(* Schneider Machine Expert - Basic project scelta_strategia_meccanismo, file version 3.0.0.0 *)
(* ProjectInformations: Name=Nuovo progetto *)

HARDWARE
  Cpu 0: TM221CE40R
  EthernetConfiguration: NetworkName=M221, IpAllocationMode=FixedAddress, IpAddress=0.0.0.0, SubnetMask=0.0.0.0
  SerialLineConfiguration: Baud=Baud19200, Parity=ParityEven, DataBits=DataBits8, StopBits=StopBits1, PhysicalMedium=PhysicalMediumRs485, TransmissionMode=TransmissionModeModbusRtu, SlaveId=1, Addressing=SlaveAddressing
  MastTask: UsePeriodScanMode=false, PeriodScan=100
  FastTask: Period=255
  CpuBehavior: StartingMode=StartAsPreviousState, AutoSaveRamOnEeprom=true, WatchdogPeriod=250

SYMBOLS  (address, symbol, comment, settings)
  %M5         "placeholder"
  %MW0      CONTA_PIU_UNDICI
  %MW1      CONTA_PIU_DODICI
  %MW2      CONTA_PIU_TREDICI
  %C0       CONTATORE  [Preset=100]
  %IW0.0    STRATEGIA  "11 = più undici; 12 = più dodici; 13 = più tredici;"  [Type=Type_0_10V, Scope=Scope_Normal, Minimum=0, Maximum=1000]

POU Nuovo POU
  (* SectionNumber=1 *)

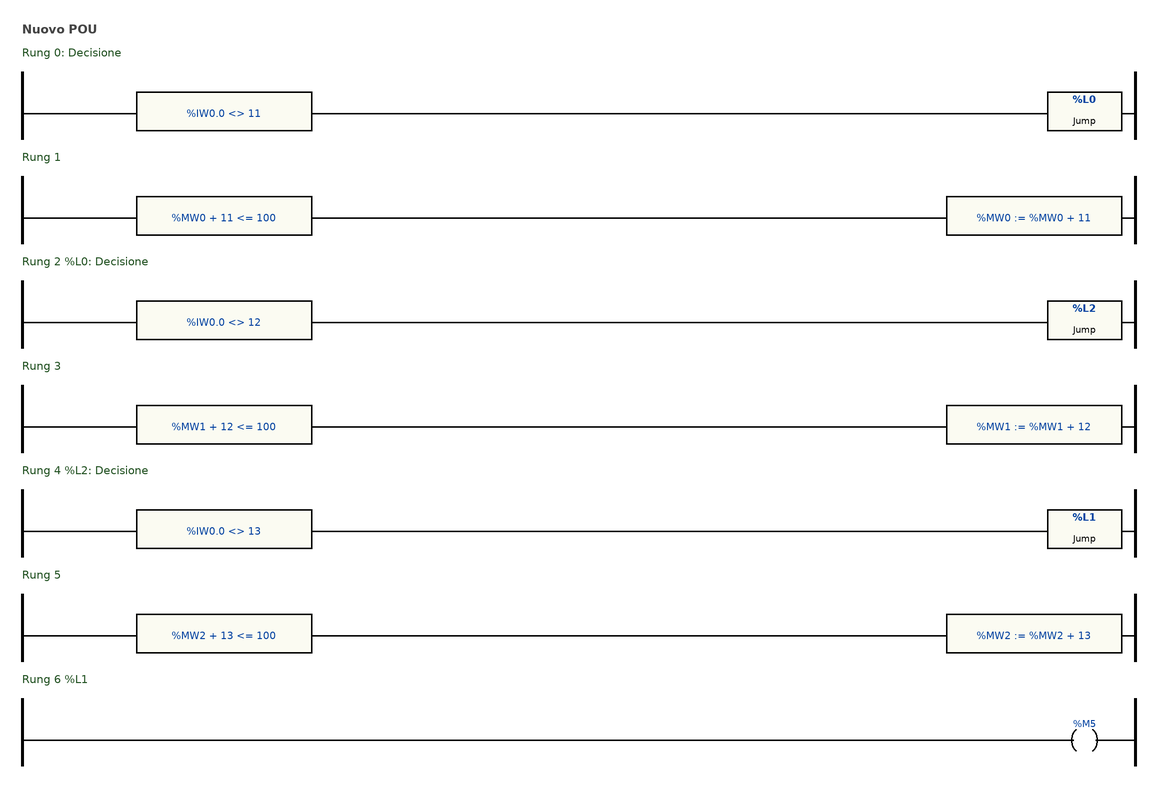

// Rung 0: Decisione
  LD [ %IW0.0 <> 11 ]     (* STRATEGIA *)
  JMPC %L0
  // as ST:
  //   IF STRATEGIA <> 11 THEN JMP %L0; END_IF;

// Rung 1
  LD 1
  AND [ %MW0 + 11 <= 100 ](* CONTA_PIU_UNDICI *)
  [ %MW0 := %MW0 + 11 ]   (* CONTA_PIU_UNDICI, CONTA_PIU_UNDICI *)
  // as ST:
  //   IF CONTA_PIU_UNDICI + 11 <= 100 THEN CONTA_PIU_UNDICI := CONTA_PIU_UNDICI + 11; END_IF;

// Rung 2 %L0: Decisione
  %L0:
  LD [ %IW0.0 <> 12 ]     (* STRATEGIA *)
  JMPC %L2
  // as ST:
  //   %L0:
  //   IF STRATEGIA <> 12 THEN JMP %L2; END_IF;

// Rung 3
  LD 1
  AND [ %MW1 + 12 <= 100 ](* CONTA_PIU_DODICI *)
  [ %MW1 := %MW1 + 12 ]   (* CONTA_PIU_DODICI, CONTA_PIU_DODICI *)
  // as ST:
  //   IF CONTA_PIU_DODICI + 12 <= 100 THEN CONTA_PIU_DODICI := CONTA_PIU_DODICI + 12; END_IF;

// Rung 4 %L2: Decisione
  %L2:
  LD [ %IW0.0 <> 13 ]     (* STRATEGIA *)
  JMPC %L1
  // as ST:
  //   %L2:
  //   IF STRATEGIA <> 13 THEN JMP %L1; END_IF;

// Rung 5
  LD 1
  AND [ %MW2 + 13 <= 100 ](* CONTA_PIU_TREDICI *)
  [ %MW2 := %MW2 + 13 ]   (* CONTA_PIU_TREDICI, CONTA_PIU_TREDICI *)
  // as ST:
  //   IF CONTA_PIU_TREDICI + 13 <= 100 THEN CONTA_PIU_TREDICI := CONTA_PIU_TREDICI + 13; END_IF;

// Rung 6 %L1
  %L1:
  LD 1
  ST %M5
  // as ST:
  //   %L1:
  //   %M5 := TRUE;
